// TIA Portal V20 export
DATA_BLOCK "DB_IO_Runtime"   // DB811
TITLE = DB_IO_Runtime
{ S7_Optimized_Access := 'FALSE' }
VERSION : 0.1
// IO test runtime DB811 non-optimized
// stored: AutoNumber false, IsOnlyStoredInLoadMemory false, IsWriteProtectedInAS false
   VAR
      DQ_Force : Array[1..20] of DWORD;
      AQ_mA : Array[1..160] of Real;
      Heartbeat : UInt;
   END_VAR
BEGIN
END_DATA_BLOCK
